Staubli VAL3: remErrInvalid.pgx

program remErrInvalid(string sCmd (dimensions=1), string& sArgs[] (dimensions=1), string& sReturn[] (dimensions=1))
begin
  // Error raised when an invalid string argument is recieved
  //
  logMsg("call remErrInvalid")
  sReturn="ERROR 104"
  sReturn=sReturn+": "+sCmd
  sReturn=sReturn+" recieved invalid string arg "
  sReturn=sReturn+sArgs+"."
  putln(sReturn)
  logMsg(sReturn)
end
